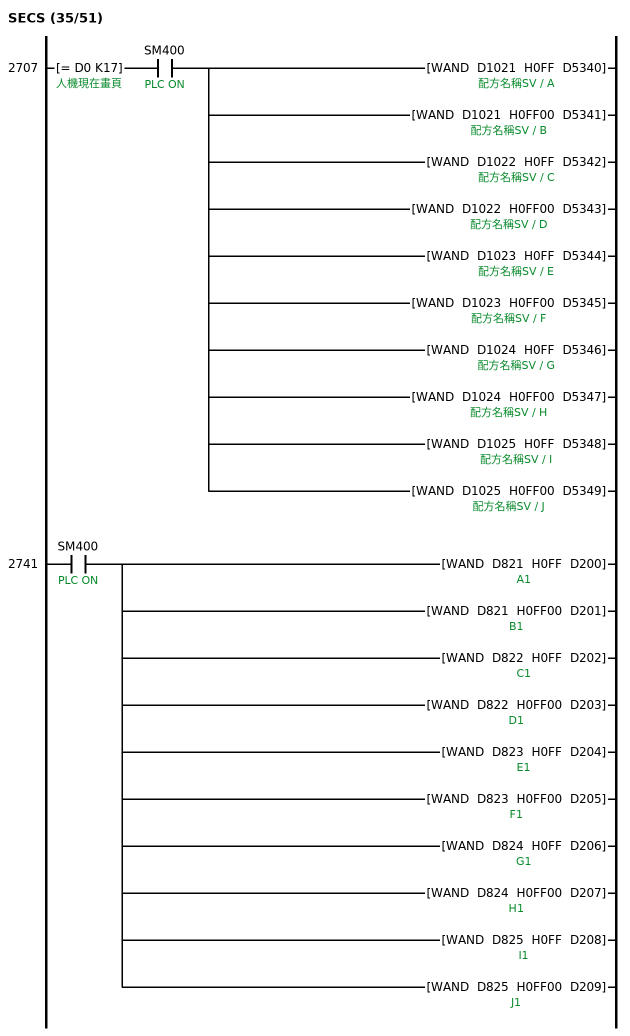
2707  LD=     D0 K17  ; 人機現在畫頁
      AND     SM400  ; PLC ON
      WAND    D1021 H0FF D5340  ; A
      WAND    D1021 H0FF00 D5341  ; B
      WAND    D1022 H0FF D5342  ; 配方名稱SV / C
      WAND    D1022 H0FF00 D5343  ; D
      WAND    D1023 H0FF D5344  ; 配方名稱SV / E
      WAND    D1023 H0FF00 D5345  ; F
      WAND    D1024 H0FF D5346  ; 配方名稱SV / G
      WAND    D1024 H0FF00 D5347  ; H
      WAND    D1025 H0FF D5348  ; 配方名稱SV / I
      WAND    D1025 H0FF00 D5349  ; J
2741  LD      SM400  ; PLC ON
      WAND    D821 H0FF D200  ; A1
      WAND    D821 H0FF00 D201  ; B1
      WAND    D822 H0FF D202  ; C1
      WAND    D822 H0FF00 D203  ; D1
      WAND    D823 H0FF D204  ; E1
      WAND    D823 H0FF00 D205  ; F1
      WAND    D824 H0FF D206  ; G1
      WAND    D824 H0FF00 D207  ; H1
      WAND    D825 H0FF D208  ; I1
      WAND    D825 H0FF00 D209  ; J1
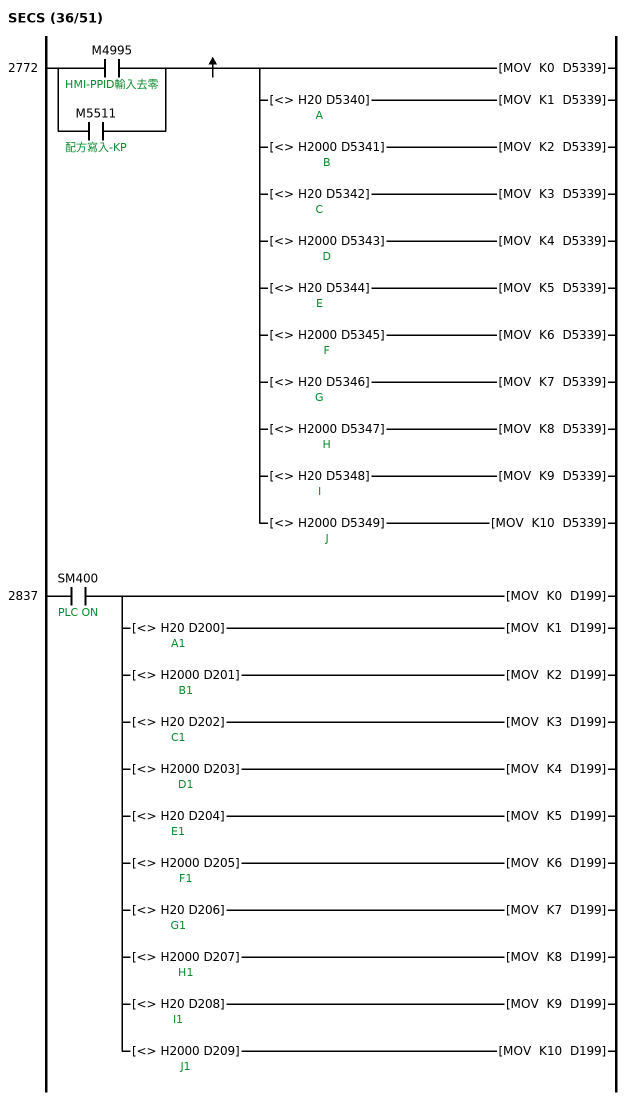
2772  LD      M4995  ; HMI-PPID輸入去零
      OR      M5511  ; 配方寫入-KP
      MEP
      MOV     K0 D5339
      MPS
      AND<>   H20 D5340  ; A
      MOV     K1 D5339
      MRD
      AND<>   H2000 D5341  ; B
      MOV     K2 D5339
      MRD
      AND<>   H20 D5342  ; C
      MOV     K3 D5339
      MRD
      AND<>   H2000 D5343  ; D
      MOV     K4 D5339
      MRD
      AND<>   H20 D5344  ; E
      MOV     K5 D5339
      MRD
      AND<>   H2000 D5345  ; F
      MOV     K6 D5339
      MRD
      AND<>   H20 D5346  ; G
      MOV     K7 D5339
      MRD
      AND<>   H2000 D5347  ; H
      MOV     K8 D5339
      MRD
      AND<>   H20 D5348  ; I
      MOV     K9 D5339
      MPP
      AND<>   H2000 D5349  ; J
      MOV     K10 D5339
2837  LD      SM400  ; PLC ON
      MOV     K0 D199
      MPS
      AND<>   H20 D200  ; A1
      MOV     K1 D199
      MRD
      AND<>   H2000 D201  ; B1
      MOV     K2 D199
      MRD
      AND<>   H20 D202  ; C1
      MOV     K3 D199
      MRD
      AND<>   H2000 D203  ; D1
      MOV     K4 D199
      MRD
      AND<>   H20 D204  ; E1
      MOV     K5 D199
      MRD
      AND<>   H2000 D205  ; F1
      MOV     K6 D199
      MRD
      AND<>   H20 D206  ; G1
      MOV     K7 D199
      MRD
      AND<>   H2000 D207  ; H1
      MOV     K8 D199
      MRD
      AND<>   H20 D208  ; I1
      MOV     K9 D199
      MPP
      AND<>   H2000 D209  ; J1
      MOV     K10 D199
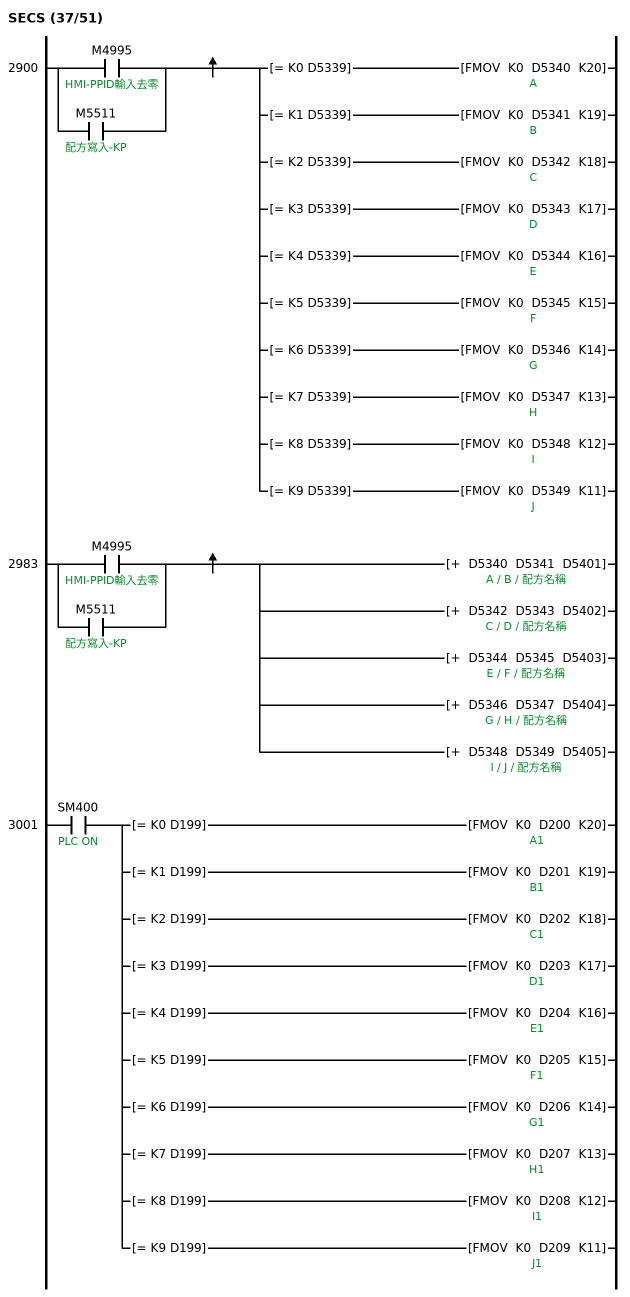
2900  LD      M4995  ; HMI-PPID輸入去零
      OR      M5511  ; 配方寫入-KP
      MEP
      MPS
      AND=    K0 D5339
      FMOV    K0 D5340 K20
      MRD
      AND=    K1 D5339
      FMOV    K0 D5341 K19
      MRD
      AND=    K2 D5339
      FMOV    K0 D5342 K18
      MRD
      AND=    K3 D5339
      FMOV    K0 D5343 K17
      MRD
      AND=    K4 D5339
      FMOV    K0 D5344 K16
      MRD
      AND=    K5 D5339
      FMOV    K0 D5345 K15
      MRD
      AND=    K6 D5339
      FMOV    K0 D5346 K14
      MRD
      AND=    K7 D5339
      FMOV    K0 D5347 K13
      MRD
      AND=    K8 D5339
      FMOV    K0 D5348 K12
      MPP
      AND=    K9 D5339
      FMOV    K0 D5349 K11
2983  LD      M4995  ; HMI-PPID輸入去零
      OR      M5511  ; 配方寫入-KP
      MEP
      +       D5340 D5341 D5401
      +       D5342 D5343 D5402  ; 配方名稱
      +       D5344 D5345 D5403  ; 配方名稱
      +       D5346 D5347 D5404  ; 配方名稱
      +       D5348 D5349 D5405  ; 配方名稱
3001  LD      SM400  ; PLC ON
      MPS
      AND=    K0 D199
      FMOV    K0 D200 K20
      MRD
      AND=    K1 D199
      FMOV    K0 D201 K19
      MRD
      AND=    K2 D199
      FMOV    K0 D202 K18
      MRD
      AND=    K3 D199
      FMOV    K0 D203 K17
      MRD
      AND=    K4 D199
      FMOV    K0 D204 K16
      MRD
      AND=    K5 D199
      FMOV    K0 D205 K15
      MRD
      AND=    K6 D199
      FMOV    K0 D206 K14
      MRD
      AND=    K7 D199
      FMOV    K0 D207 K13
      MRD
      AND=    K8 D199
      FMOV    K0 D208 K12
      MPP
      AND=    K9 D199
      FMOV    K0 D209 K11
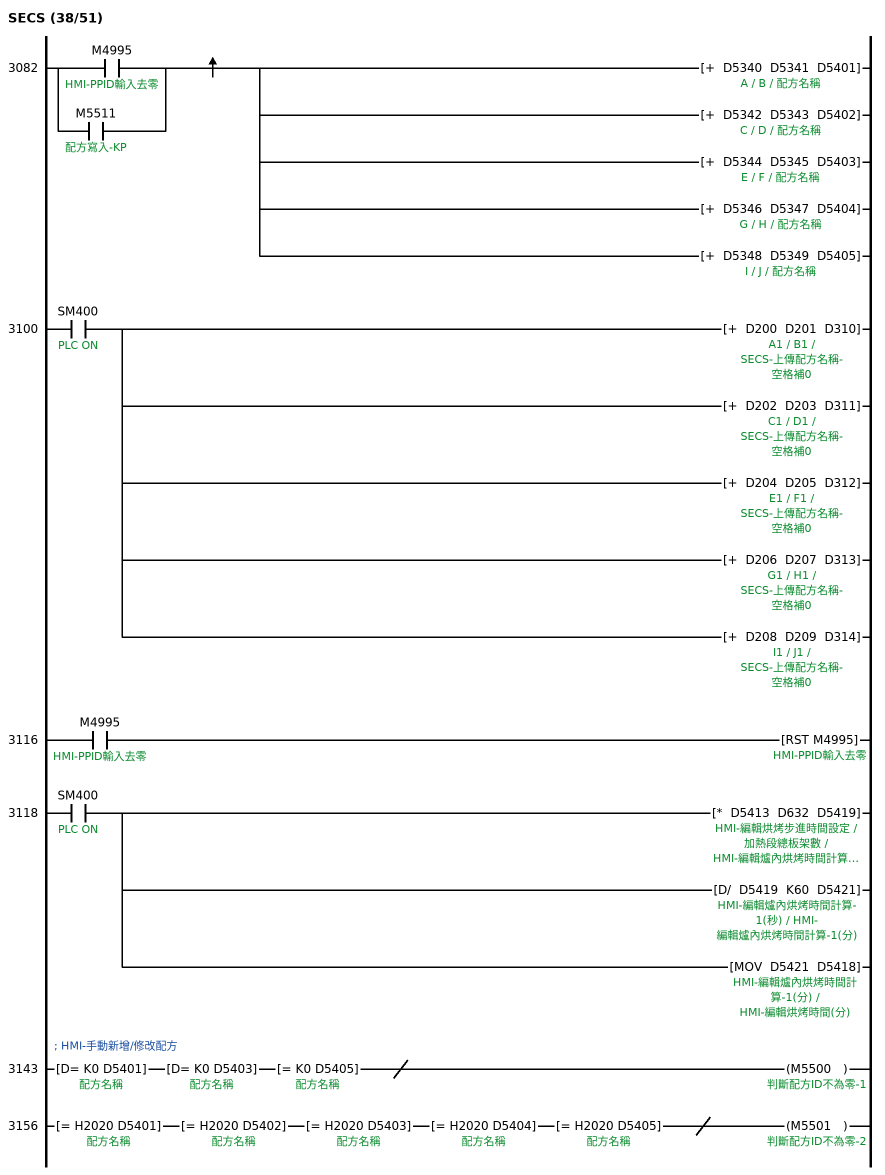
3082  LD      M4995  ; HMI-PPID輸入去零
      OR      M5511  ; 配方寫入-KP
      MEP
      +       D5340 D5341 D5401
      +       D5342 D5343 D5402
      +       D5344 D5345 D5403
      +       D5346 D5347 D5404
      +       D5348 D5349 D5405
3100  LD      SM400  ; PLC ON
      +       D200 D201 D310  ; SECS-上傳配方名稱-空格補0
      +       D202 D203 D311  ; SECS-上傳配方名稱-空格補0
      +       D204 D205 D312  ; SECS-上傳配方名稱-空格補0
      +       D206 D207 D313  ; SECS-上傳配方名稱-空格補0
      +       D208 D209 D314  ; SECS-上傳配方名稱-空格補0
3116  LD      M4995  ; HMI-PPID輸入去零
      RST     M4995  ; HMI-PPID輸入去零
3118  LD      SM400  ; PLC ON
      *       D5413 D632 D5419  ; HMI-編輯烘烤步進時間設定 / 加熱段總板架數 / HMI-編輯爐內烘烤時間計算-1(秒)
      D/      D5419 K60 D5421  ; HMI-編輯爐內烘烤時間計算-1(分)
      MOV     D5421 D5418  ; HMI-編輯烘烤時間(分)
; HMI-手動新增/修改配方
3143  LDD=    K0 D5401  ; 配方名稱
      ANDD=   K0 D5403  ; 配方名稱
      AND=    K0 D5405  ; 配方名稱
      INV
      OUT     M5500  ; 判斷配方ID不為零-1
3156  LD=     H2020 D5401  ; 配方名稱
      AND=    H2020 D5402  ; 配方名稱
      AND=    H2020 D5403  ; 配方名稱
      AND=    H2020 D5404  ; 配方名稱
      AND=    H2020 D5405  ; 配方名稱
      INV
      OUT     M5501  ; 判斷配方ID不為零-2
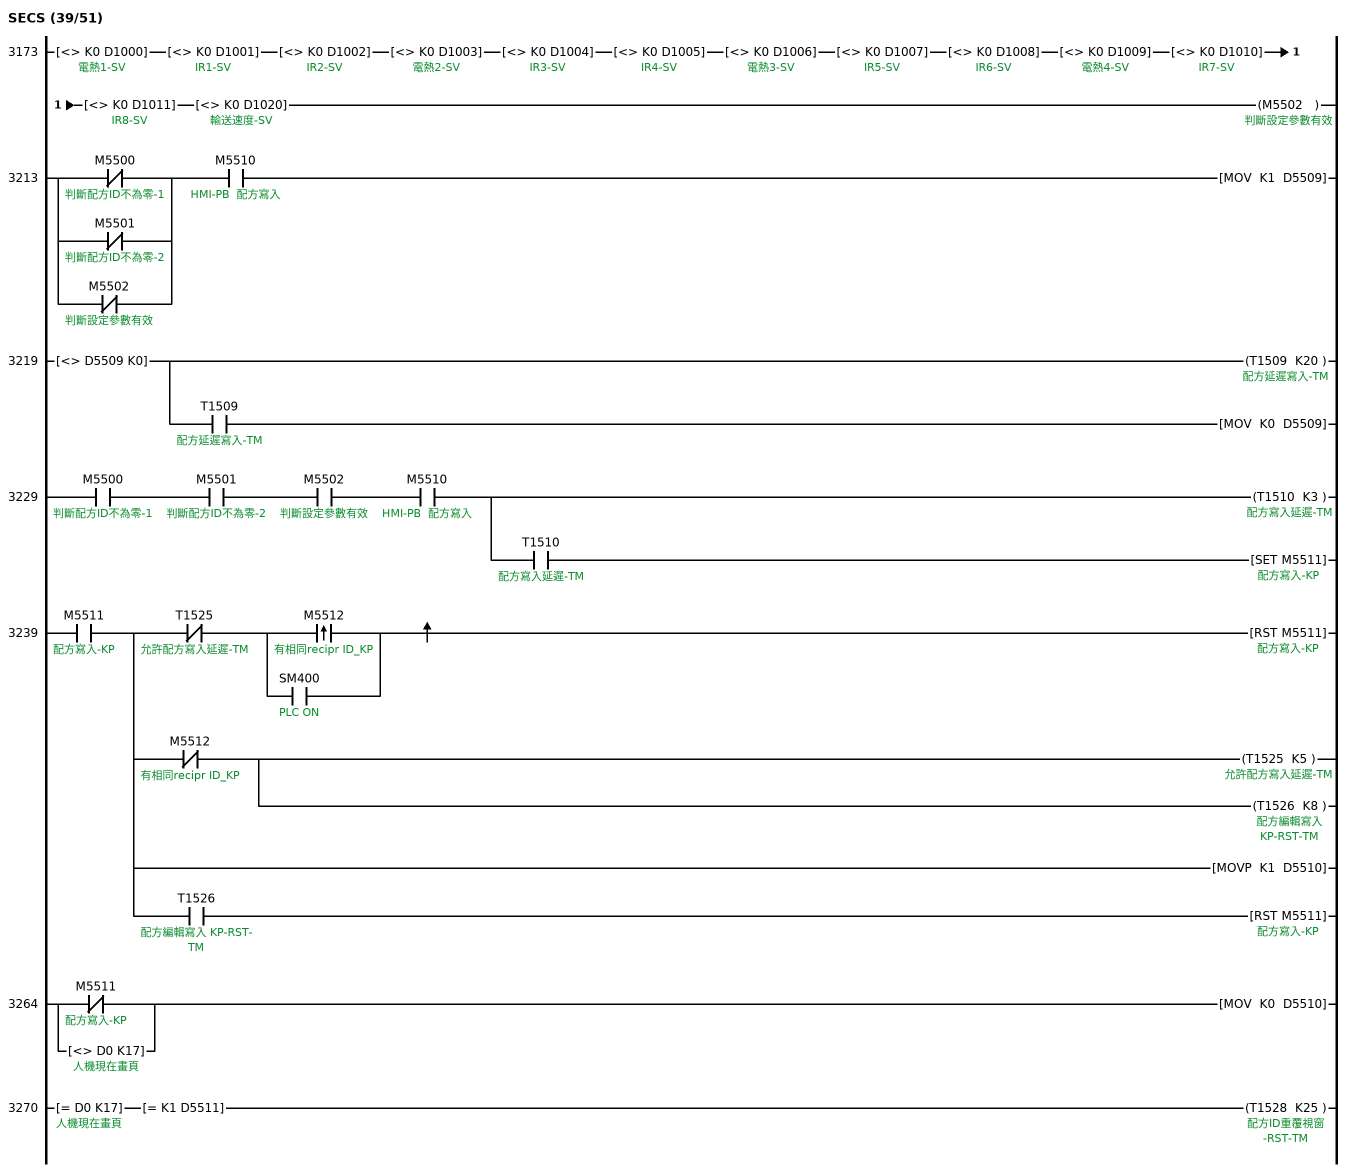
3173  LD<>    K0 D1000  ; 電熱1-SV
      AND<>   K0 D1001  ; IR1-SV
      AND<>   K0 D1002  ; IR2-SV
      AND<>   K0 D1003  ; 電熱2-SV
      AND<>   K0 D1004  ; IR3-SV
      AND<>   K0 D1005  ; IR4-SV
      AND<>   K0 D1006  ; 電熱3-SV
      AND<>   K0 D1007  ; IR5-SV
      AND<>   K0 D1008  ; IR6-SV
      AND<>   K0 D1009  ; 電熱4-SV
      AND<>   K0 D1010  ; IR7-SV
      AND<>   K0 D1011  ; IR8-SV
      AND<>   K0 D1020  ; 輸送速度-SV
      OUT     M5502  ; 判斷設定參數有效
3213  LDI     M5500  ; 判斷配方ID不為零-1
      ORI     M5501  ; 判斷配方ID不為零-2
      ORI     M5502  ; 判斷設定參數有效
      AND     M5510  ; HMI-PB  配方寫入
      MOV     K1 D5509
3219  LD<>    D5509 K0
      OUT     T1509 K20  ; 配方延遲寫入-TM
      AND     T1509  ; 配方延遲寫入-TM
      MOV     K0 D5509
3229  LD      M5500  ; 判斷配方ID不為零-1
      AND     M5501  ; 判斷配方ID不為零-2
      AND     M5502  ; 判斷設定參數有效
      AND     M5510  ; HMI-PB  配方寫入
      OUT     T1510 K3  ; 配方寫入延遲-TM
      AND     T1510  ; 配方寫入延遲-TM
      SET     M5511  ; 配方寫入-KP
3239  LD      M5511  ; 配方寫入-KP
      MPS
      ANI     T1525  ; 允許配方寫入延遲-TM
      LDP     M5512  ; 有相同recipr ID_KP
      OR      SM400  ; PLC ON
      ANB
      MEP
      RST     M5511  ; 配方寫入-KP
      MRD
      ANI     M5512  ; 有相同recipr ID_KP
      OUT     T1525 K5  ; 允許配方寫入延遲-TM
      OUT     T1526 K8  ; 配方編輯寫入 KP-RST-TM
      MPP
      MOVP    K1 D5510
      AND     T1526  ; 配方編輯寫入 KP-RST-TM
      RST     M5511  ; 配方寫入-KP
3264  LDI     M5511  ; 配方寫入-KP
      OR<>    D0 K17  ; 人機現在畫頁
      MOV     K0 D5510
3270  LD=     D0 K17  ; 人機現在畫頁
      AND=    K1 D5511
      OUT     T1528 K25  ; 配方ID重覆視窗  -RST-TM
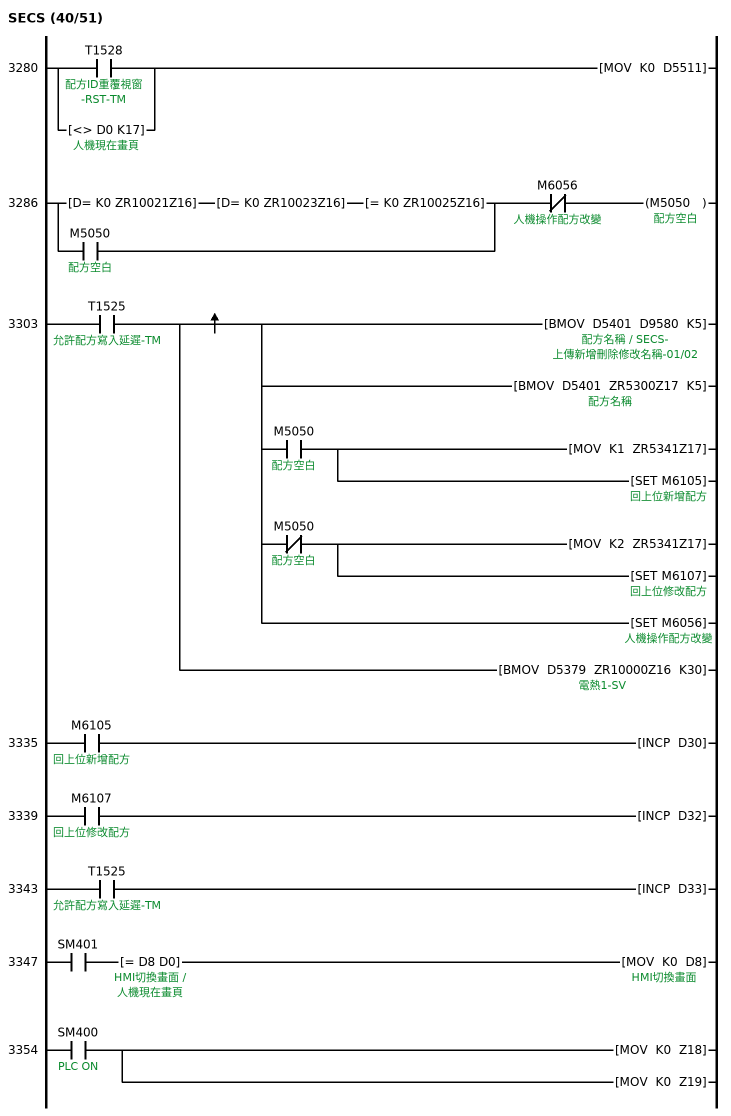
3280  LD      T1528  ; 配方ID重覆視窗  -RST-TM
      OR<>    D0 K17  ; 人機現在畫頁
      MOV     K0 D5511
3286  LDD=    K0 ZR10021Z16
      ANDD=   K0 ZR10023Z16
      AND=    K0 ZR10025Z16
      OR      M5050  ; 配方空白
      ANI     M6056  ; 人機操作配方改變
      OUT     M5050  ; 配方空白
3303  LD      T1525  ; 允許配方寫入延遲-TM
      MPS
      MEP
      BMOV    D5401 D9580 K5  ; SECS-上傳新增刪除修改名稱-01/02
      BMOV    D5401 ZR5300Z17 K5
      MPS
      AND     M5050  ; 配方空白
      MOV     K1 ZR5341Z17
      SET     M6105  ; 回上位新增配方
      MRD
      ANI     M5050  ; 配方空白
      MOV     K2 ZR5341Z17
      SET     M6107  ; 回上位修改配方
      MPP
      SET     M6056  ; 人機操作配方改變
      MPP
      BMOV    D5379 ZR10000Z16 K30
3335  LD      M6105  ; 回上位新增配方
      INCP    D30
3339  LD      M6107  ; 回上位修改配方
      INCP    D32
3343  LD      T1525  ; 允許配方寫入延遲-TM
      INCP    D33
3347  LD      SM401
      AND=    D8 D0  ; HMI切換畫面 / 人機現在畫頁
      MOV     K0 D8
3354  LD      SM400  ; PLC ON
      MOV     K0 Z18
      MOV     K0 Z19
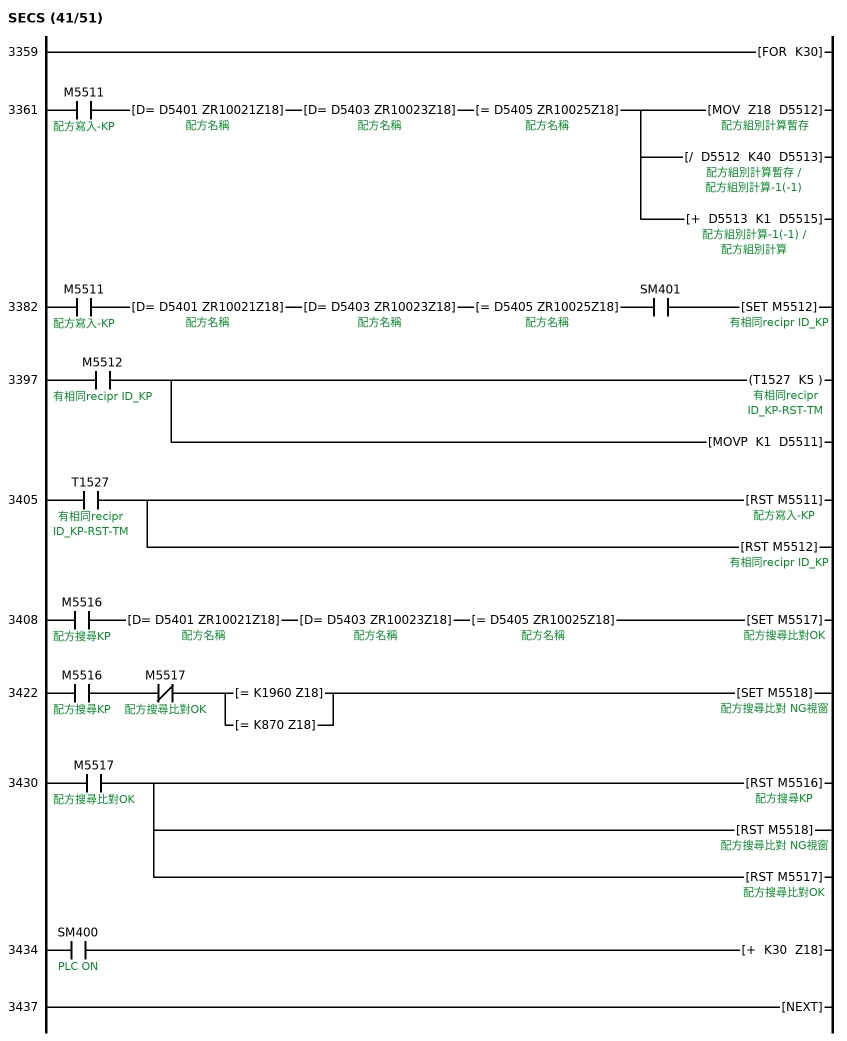
3359  FOR     K30
3361  LD      M5511  ; 配方寫入-KP
      ANDD=   D5401 ZR10021Z18  ; 配方名稱
      ANDD=   D5403 ZR10023Z18  ; 配方名稱
      AND=    D5405 ZR10025Z18  ; 配方名稱
      MOV     Z18 D5512  ; 配方組別計算暫存
      /       D5512 K40 D5513  ; 配方組別計算-1(-1)
      +       D5513 K1 D5515  ; 配方組別計算
3382  LD      M5511  ; 配方寫入-KP
      ANDD=   D5401 ZR10021Z18  ; 配方名稱
      ANDD=   D5403 ZR10023Z18  ; 配方名稱
      AND=    D5405 ZR10025Z18  ; 配方名稱
      AND     SM401
      SET     M5512  ; 有相同recipr ID_KP
3397  LD      M5512  ; 有相同recipr ID_KP
      OUT     T1527 K5  ; 有相同recipr ID_KP-RST-TM
      MOVP    K1 D5511
3405  LD      T1527  ; 有相同recipr ID_KP-RST-TM
      RST     M5511  ; 配方寫入-KP
      RST     M5512  ; 有相同recipr ID_KP
3408  LD      M5516  ; 配方搜尋KP
      ANDD=   D5401 ZR10021Z18  ; 配方名稱
      ANDD=   D5403 ZR10023Z18  ; 配方名稱
      AND=    D5405 ZR10025Z18  ; 配方名稱
      SET     M5517  ; 配方搜尋比對OK
3422  LD      M5516  ; 配方搜尋KP
      ANI     M5517  ; 配方搜尋比對OK
      LD=     K1960 Z18
      OR=     K870 Z18
      ANB
      SET     M5518  ; 配方搜尋比對 NG視窗
3430  LD      M5517  ; 配方搜尋比對OK
      RST     M5516  ; 配方搜尋KP
      RST     M5518  ; 配方搜尋比對 NG視窗
      RST     M5517  ; 配方搜尋比對OK
3434  LD      SM400  ; PLC ON
      +       K30 Z18
3437  NEXT
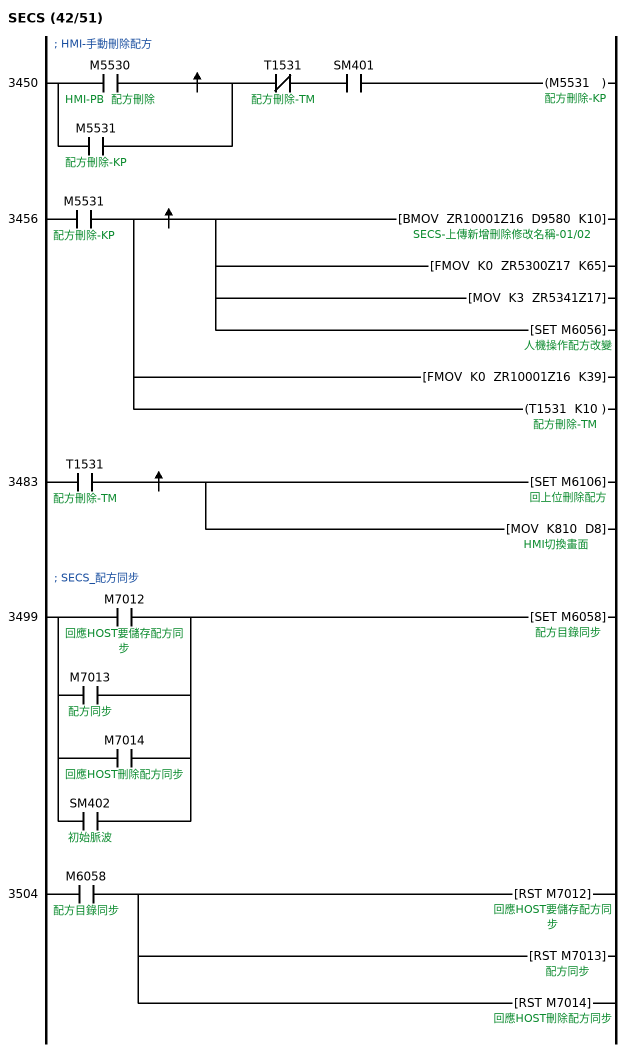
; HMI-手動刪除配方
3450  LD      M5530  ; HMI-PB  配方刪除
      MEP
      OR      M5531  ; 配方刪除-KP
      ANI     T1531  ; 配方刪除-TM
      AND     SM401
      OUT     M5531  ; 配方刪除-KP
3456  LD      M5531  ; 配方刪除-KP
      MPS
      MEP
      BMOV    ZR10001Z16 D9580 K10
      FMOV    K0 ZR5300Z17 K65
      MOV     K3 ZR5341Z17
      SET     M6056  ; 人機操作配方改變
      MPP
      FMOV    K0 ZR10001Z16 K39
      OUT     T1531 K10  ; 配方刪除-TM
3483  LD      T1531  ; 配方刪除-TM
      MEP
      SET     M6106  ; 回上位刪除配方
      MOV     K810 D8
; SECS_配方同步
3499  LD      M7012  ; 回應HOST要儲存配方同步
      OR      M7013  ; 配方同步
      OR      M7014  ; 回應HOST刪除配方同步
      OR      SM402  ; 初始脈波
      SET     M6058  ; 配方目錄同步
3504  LD      M6058  ; 配方目錄同步
      RST     M7012  ; 回應HOST要儲存配方同步
      RST     M7013  ; 配方同步
      RST     M7014  ; 回應HOST刪除配方同步
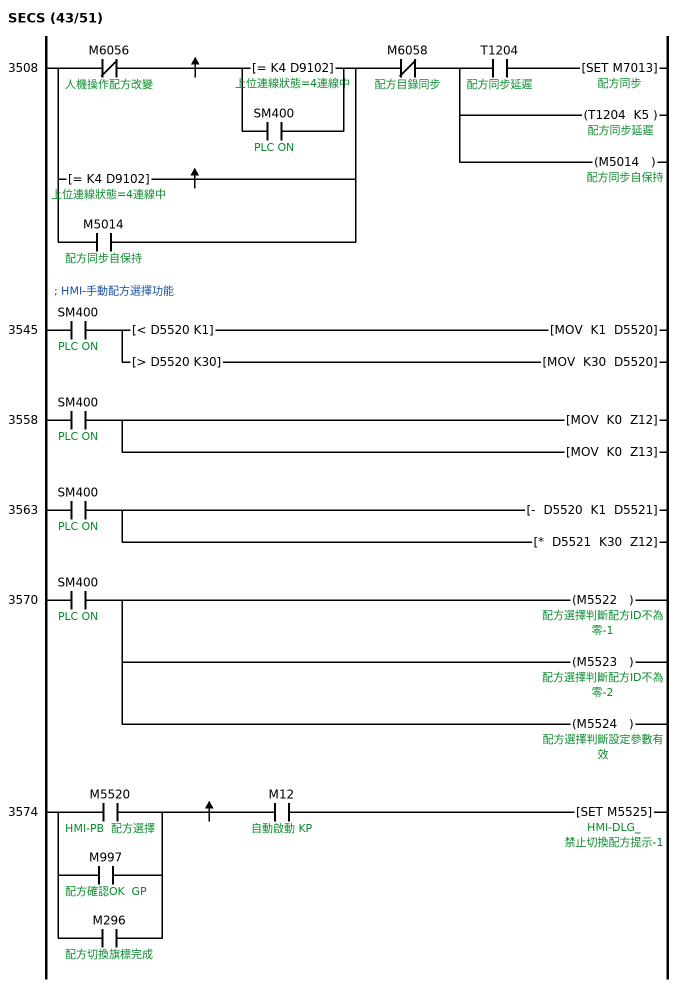
3508  LDI     M6056  ; 人機操作配方改變
      MEP
      LD=     K4 D9102  ; 上位連線狀態=4連線中
      OR      SM400  ; PLC ON
      ANB
      LD=     K4 D9102  ; 上位連線狀態=4連線中
      MEP
      ORB
      OR      M5014  ; 配方同步自保持
      ANI     M6058  ; 配方目錄同步
      MPS
      AND     T1204  ; 配方同步延遲
      SET     M7013  ; 配方同步
      MPP
      OUT     T1204 K5  ; 配方同步延遲
      OUT     M5014  ; 配方同步自保持
; HMI-手動配方選擇功能
3545  LD      SM400  ; PLC ON
      MPS
      AND<    D5520 K1
      MOV     K1 D5520
      MPP
      AND>    D5520 K30
      MOV     K30 D5520
3558  LD      SM400  ; PLC ON
      MOV     K0 Z12
      MOV     K0 Z13
3563  LD      SM400  ; PLC ON
      -       D5520 K1 D5521
      *       D5521 K30 Z12
3570  LD      SM400  ; PLC ON
      OUT     M5522  ; 配方選擇判斷配方ID不為零-1
      OUT     M5523  ; 配方選擇判斷配方ID不為零-2
      OUT     M5524  ; 配方選擇判斷設定參數有效
3574  LD      M5520  ; HMI-PB  配方選擇
      OR      M997  ; 配方確認OK  GP
      OR      M296  ; 配方切換旗標完成
      MEP
      AND     M12  ; 自動啟動 KP
      SET     M5525  ; HMI-DLG_禁止切換配方提示-1
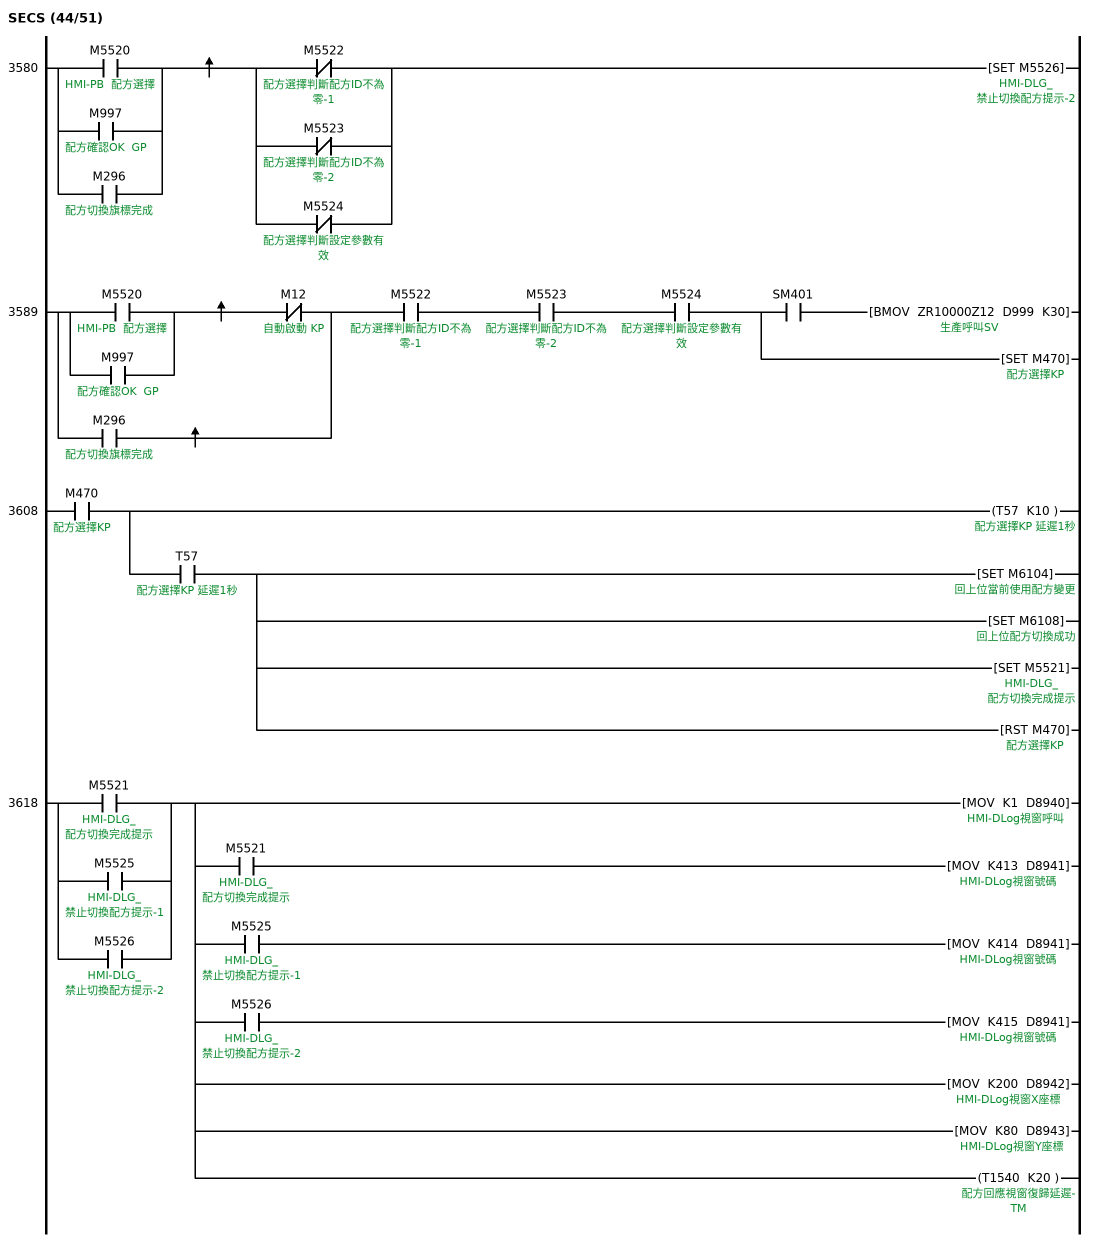
3580  LD      M5520  ; HMI-PB  配方選擇
      OR      M997  ; 配方確認OK  GP
      OR      M296  ; 配方切換旗標完成
      MEP
      LDI     M5522  ; 配方選擇判斷配方ID不為零-1
      ORI     M5523  ; 配方選擇判斷配方ID不為零-2
      ORI     M5524  ; 配方選擇判斷設定參數有效
      ANB
      SET     M5526  ; HMI-DLG_禁止切換配方提示-2
3589  LD      M5520  ; HMI-PB  配方選擇
      OR      M997  ; 配方確認OK  GP
      MEP
      ANI     M12  ; 自動啟動 KP
      LD      M296  ; 配方切換旗標完成
      MEP
      ORB
      AND     M5522  ; 配方選擇判斷配方ID不為零-1
      AND     M5523  ; 配方選擇判斷配方ID不為零-2
      AND     M5524  ; 配方選擇判斷設定參數有效
      MPS
      AND     SM401
      BMOV    ZR10000Z12 D999 K30
      MPP
      SET     M470  ; 配方選擇KP
3608  LD      M470  ; 配方選擇KP
      OUT     T57 K10  ; 配方選擇KP 延遲1秒
      AND     T57  ; 配方選擇KP 延遲1秒
      SET     M6104  ; 回上位當前使用配方變更
      SET     M6108  ; 回上位配方切換成功
      SET     M5521  ; HMI-DLG_配方切換完成提示
      RST     M470  ; 配方選擇KP
3618  LD      M5521  ; HMI-DLG_配方切換完成提示
      OR      M5525  ; HMI-DLG_禁止切換配方提示-1
      OR      M5526  ; HMI-DLG_禁止切換配方提示-2
      MOV     K1 D8940  ; HMI-DLog視窗呼叫
      MPS
      AND     M5521  ; HMI-DLG_配方切換完成提示
      MOV     K413 D8941  ; HMI-DLog視窗號碼
      MRD
      AND     M5525  ; HMI-DLG_禁止切換配方提示-1
      MOV     K414 D8941
      MRD
      AND     M5526  ; HMI-DLG_禁止切換配方提示-2
      MOV     K415 D8941
      MPP
      MOV     K200 D8942  ; HMI-DLog視窗X座標
      MOV     K80 D8943  ; HMI-DLog視窗Y座標
      OUT     T1540 K20  ; 配方回應視窗復歸延遲-TM
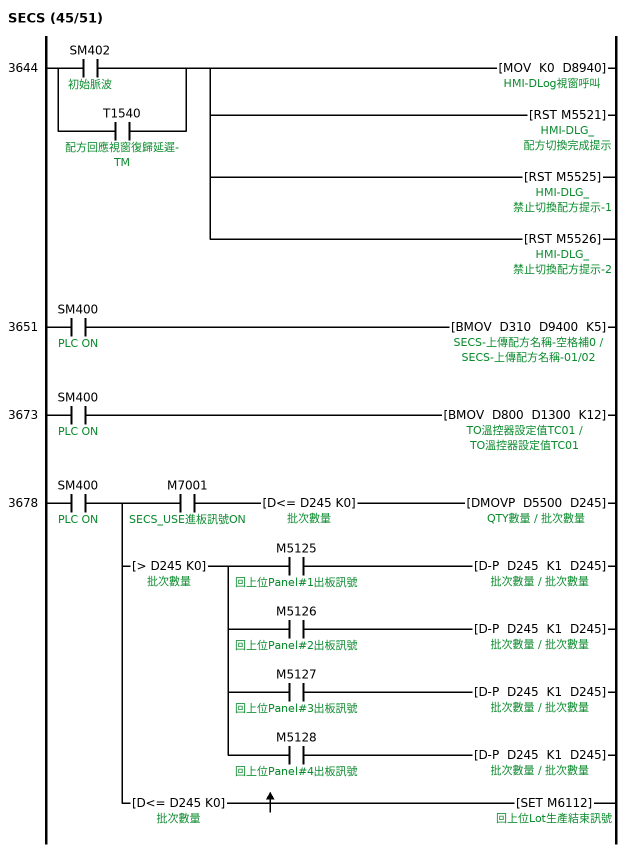
3644  LD      SM402  ; 初始脈波
      OR      T1540  ; 配方回應視窗復歸延遲-TM
      MOV     K0 D8940
      RST     M5521  ; HMI-DLG_配方切換完成提示
      RST     M5525  ; HMI-DLG_禁止切換配方提示-1
      RST     M5526  ; HMI-DLG_禁止切換配方提示-2
3651  LD      SM400  ; PLC ON
      BMOV    D310 D9400 K5  ; SECS-上傳配方名稱-01/02
        [note] D9400_上報SECS目前使用PPID名稱
3673  LD      SM400  ; PLC ON
      BMOV    D800 D1300 K12  ; TO溫控器設定值TC01
3678  LD      SM400  ; PLC ON
      MPS
      AND     M7001  ; SECS_USE進板訊號ON
      ANDD<=  D245 K0  ; 批次數量
      DMOVP   D5500 D245
      MRD
      AND>    D245 K0  ; 批次數量
      MPS
      AND     M5125  ; 回上位Panel#1出板訊號
      D-P     D245 K1 D245
      MRD
      AND     M5126  ; 回上位Panel#2出板訊號
      D-P     D245 K1 D245
      MRD
      AND     M5127  ; 回上位Panel#3出板訊號
      D-P     D245 K1 D245
      MPP
      AND     M5128  ; 回上位Panel#4出板訊號
      D-P     D245 K1 D245
      MPP
      ANDD<=  D245 K0  ; 批次數量
      MEP
      SET     M6112  ; 回上位Lot生產結束訊號
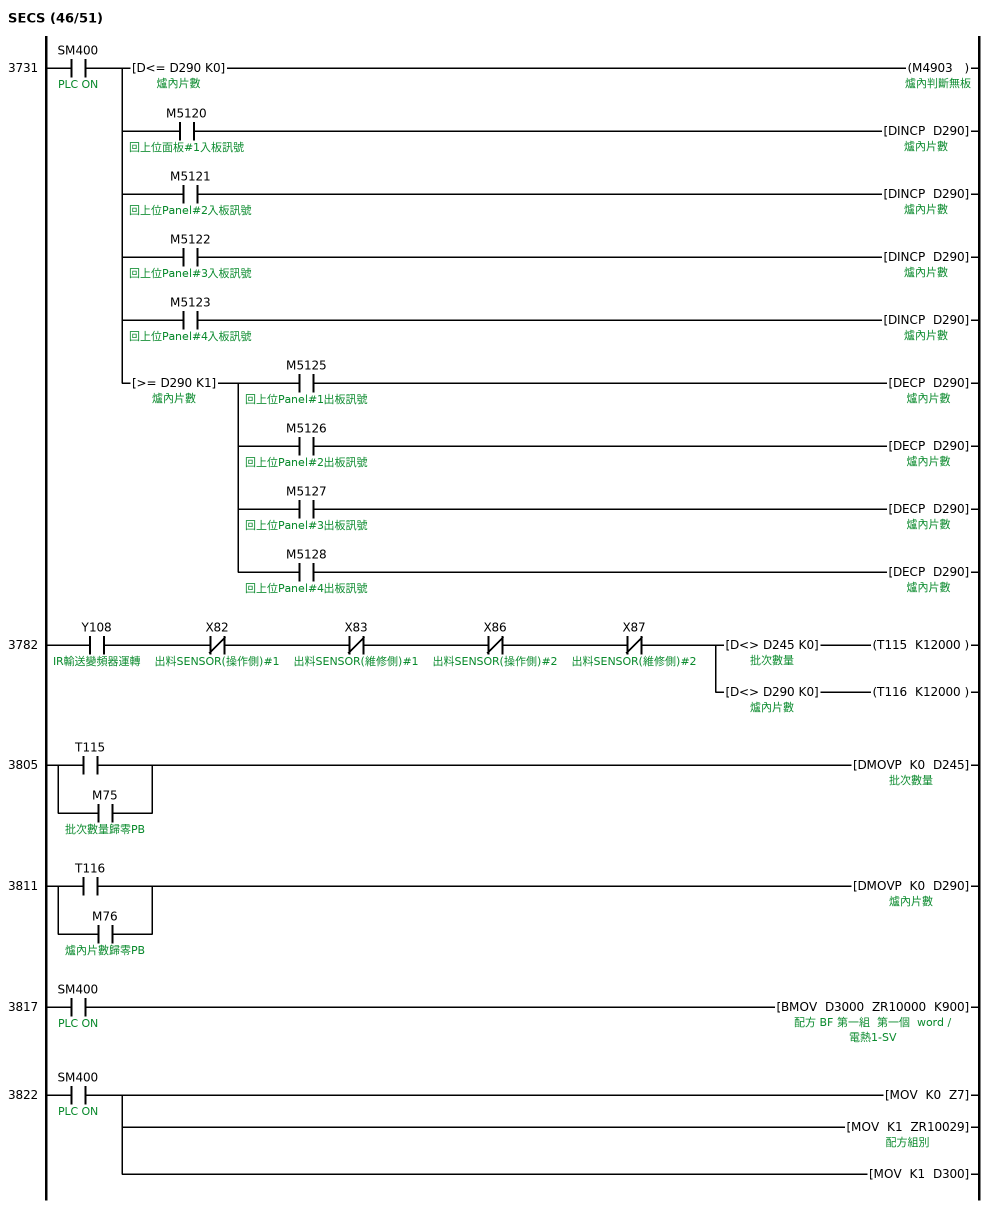
3731  LD      SM400  ; PLC ON
      MPS
      ANDD<=  D290 K0  ; 爐內片數
      OUT     M4903  ; 爐內判斷無板
      MRD
      AND     M5120  ; 回上位面板#1入板訊號
      DINCP   D290
      MRD
      AND     M5121  ; 回上位Panel#2入板訊號
      DINCP   D290
      MRD
      AND     M5122  ; 回上位Panel#3入板訊號
      DINCP   D290
      MRD
      AND     M5123  ; 回上位Panel#4入板訊號
      DINCP   D290
      MPP
      AND>=   D290 K1  ; 爐內片數
      MPS
      AND     M5125  ; 回上位Panel#1出板訊號
      DECP    D290
      MRD
      AND     M5126  ; 回上位Panel#2出板訊號
      DECP    D290
      MRD
      AND     M5127  ; 回上位Panel#3出板訊號
      DECP    D290
      MPP
      AND     M5128  ; 回上位Panel#4出板訊號
      DECP    D290
3782  LD      Y108  ; IR輸送變頻器運轉
      ANI     X82  ; 出料SENSOR(操作側)#1
      ANI     X83  ; 出料SENSOR(維修側)#1
      ANI     X86  ; 出料SENSOR(操作側)#2
      ANI     X87  ; 出料SENSOR(維修側)#2
      MPS
      ANDD<>  D245 K0  ; 批次數量
      OUT     T115 K12000
      MPP
      ANDD<>  D290 K0  ; 爐內片數
      OUT     T116 K12000
3805  LD      T115
      OR      M75  ; 批次數量歸零PB
      DMOVP   K0 D245
3811  LD      T116
      OR      M76  ; 爐內片數歸零PB
      DMOVP   K0 D290
3817  LD      SM400  ; PLC ON
      BMOV    D3000 ZR10000 K900  ; 配方 BF 第一組  第一個  word
3822  LD      SM400  ; PLC ON
      MOV     K0 Z7
      MOV     K1 ZR10029  ; 配方組別
      MOV     K1 D300
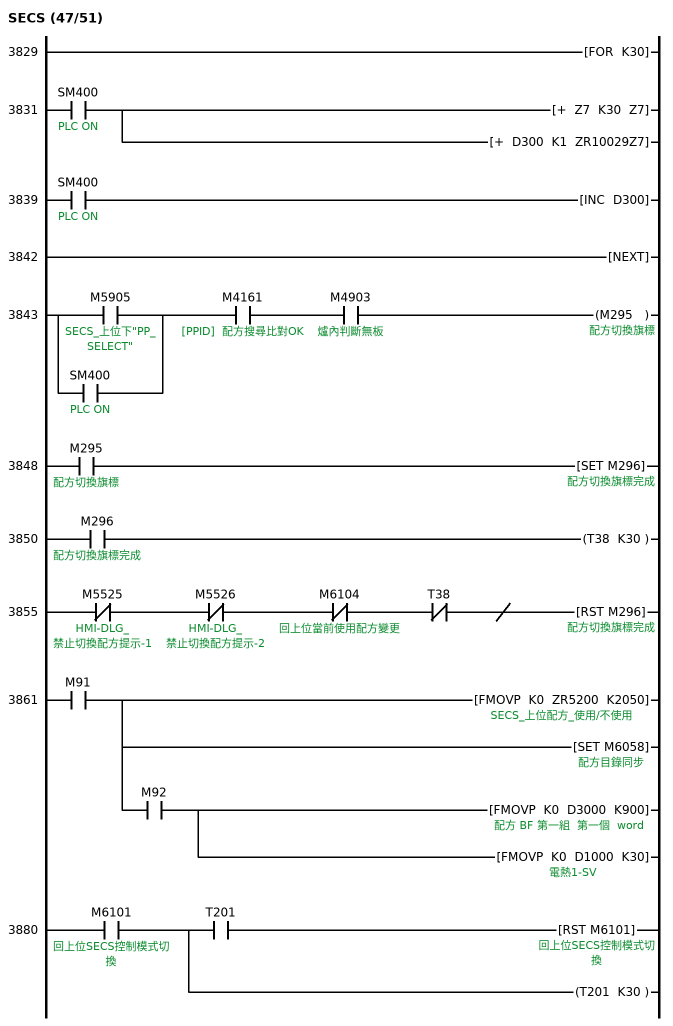
3829  FOR     K30
3831  LD      SM400  ; PLC ON
      +       Z7 K30 Z7
      +       D300 K1 ZR10029Z7
3839  LD      SM400  ; PLC ON
      INC     D300
3842  NEXT
3843  LD      M5905  ; SECS_上位下"PP_SELECT"
      OR      SM400  ; PLC ON
      AND     M4161  ; [PPID]  配方搜尋比對OK
      AND     M4903  ; 爐內判斷無板
      OUT     M295  ; 配方切換旗標
3848  LD      M295  ; 配方切換旗標
      SET     M296  ; 配方切換旗標完成
3850  LD      M296  ; 配方切換旗標完成
      OUT     T38 K30
3855  LDI     M5525  ; HMI-DLG_禁止切換配方提示-1
      ANI     M5526  ; HMI-DLG_禁止切換配方提示-2
      ANI     M6104  ; 回上位當前使用配方變更
      ANI     T38
      INV
      RST     M296  ; 配方切換旗標完成
3861  LD      M91
      FMOVP   K0 ZR5200 K2050  ; SECS_上位配方_使用/不使用
      SET     M6058  ; 配方目錄同步
      AND     M92
      FMOVP   K0 D3000 K900
      FMOVP   K0 D1000 K30
3880  LD      M6101  ; 回上位SECS控制模式切換
      MPS
      AND     T201
      RST     M6101  ; 回上位SECS控制模式切換
      MPP
      OUT     T201 K30
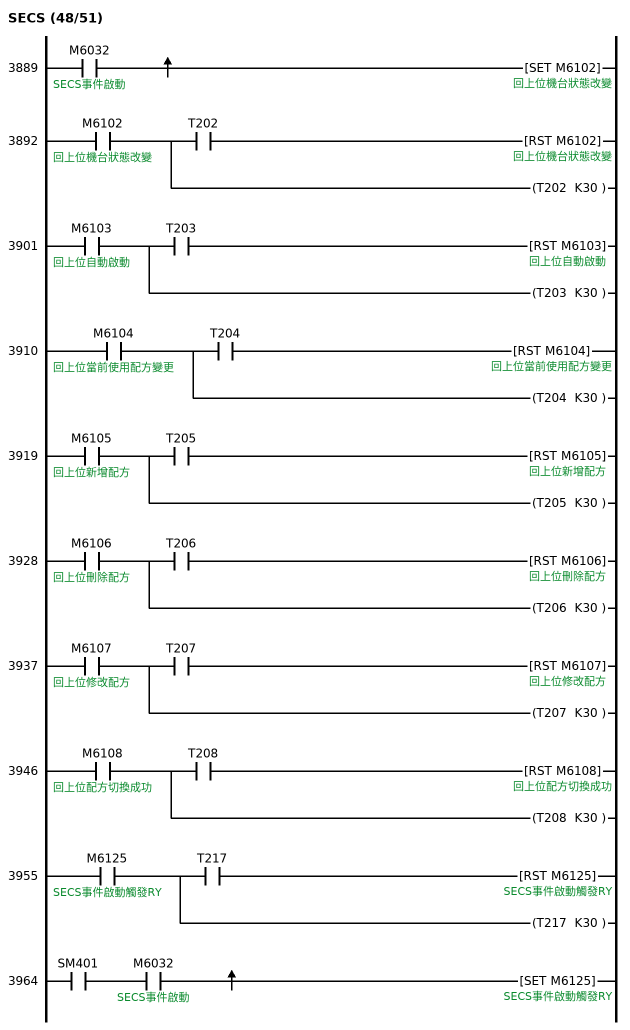
3889  LD      M6032  ; SECS事件啟動
      MEP
      SET     M6102  ; 回上位機台狀態改變
3892  LD      M6102  ; 回上位機台狀態改變
      MPS
      AND     T202
      RST     M6102  ; 回上位機台狀態改變
      MPP
      OUT     T202 K30
3901  LD      M6103  ; 回上位自動啟動
      MPS
      AND     T203
      RST     M6103  ; 回上位自動啟動
      MPP
      OUT     T203 K30
3910  LD      M6104  ; 回上位當前使用配方變更
      MPS
      AND     T204
      RST     M6104  ; 回上位當前使用配方變更
      MPP
      OUT     T204 K30
3919  LD      M6105  ; 回上位新增配方
      MPS
      AND     T205
      RST     M6105  ; 回上位新增配方
      MPP
      OUT     T205 K30
3928  LD      M6106  ; 回上位刪除配方
      MPS
      AND     T206
      RST     M6106  ; 回上位刪除配方
      MPP
      OUT     T206 K30
3937  LD      M6107  ; 回上位修改配方
      MPS
      AND     T207
      RST     M6107  ; 回上位修改配方
      MPP
      OUT     T207 K30
3946  LD      M6108  ; 回上位配方切換成功
      MPS
      AND     T208
      RST     M6108  ; 回上位配方切換成功
      MPP
      OUT     T208 K30
3955  LD      M6125  ; SECS事件啟動觸發RY
      MPS
      AND     T217
      RST     M6125  ; SECS事件啟動觸發RY
      MPP
      OUT     T217 K30
3964  LD      SM401
      AND     M6032  ; SECS事件啟動
      MEP
      SET     M6125  ; SECS事件啟動觸發RY
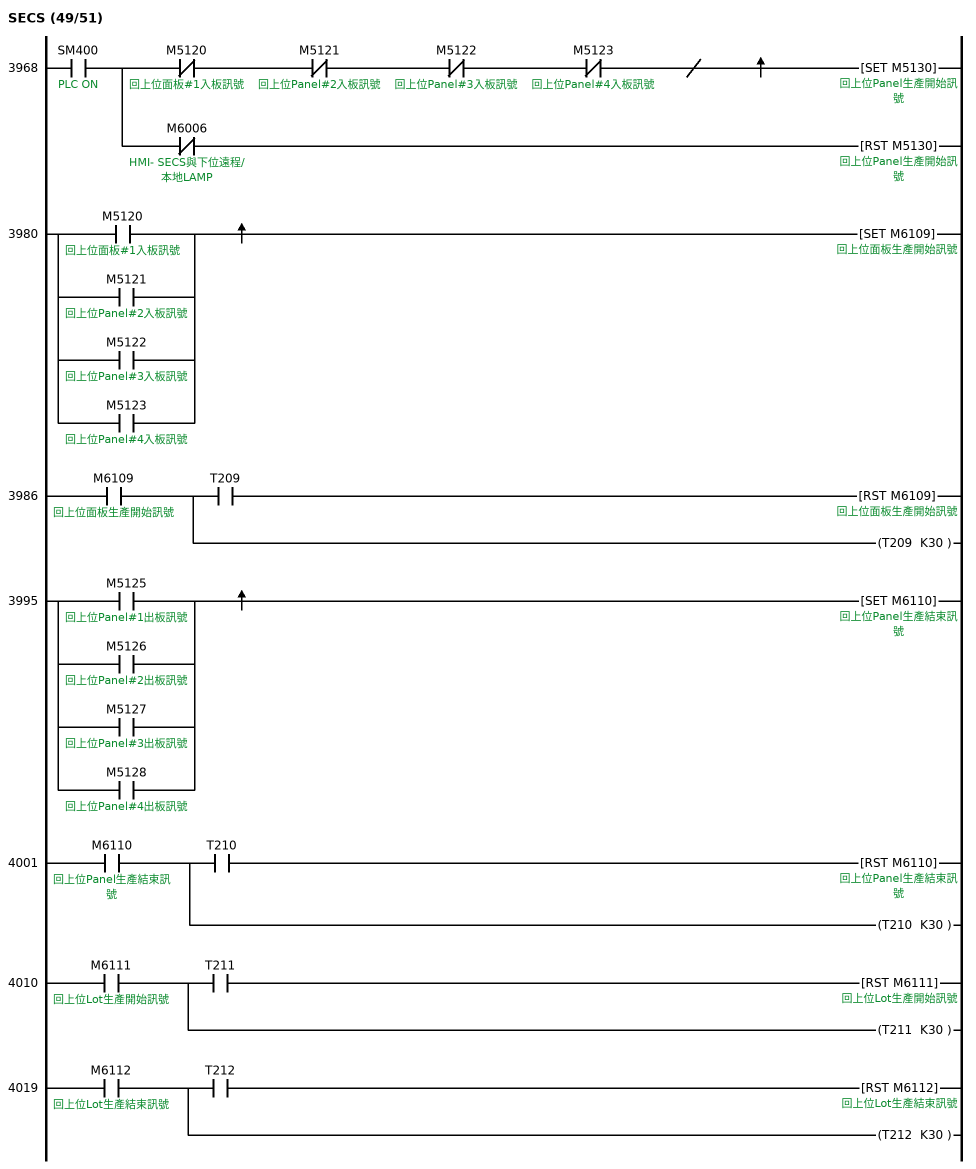
3968  LD      SM400  ; PLC ON
      MPS
      ANI     M5120  ; 回上位面板#1入板訊號
      ANI     M5121  ; 回上位Panel#2入板訊號
      ANI     M5122  ; 回上位Panel#3入板訊號
      ANI     M5123  ; 回上位Panel#4入板訊號
      INV
      MEP
      SET     M5130  ; 回上位Panel生產開始訊號
      MPP
      ANI     M6006  ; HMI- SECS與下位遠程/本地LAMP
      RST     M5130  ; 回上位Panel生產開始訊號
3980  LD      M5120  ; 回上位面板#1入板訊號
      OR      M5121  ; 回上位Panel#2入板訊號
      OR      M5122  ; 回上位Panel#3入板訊號
      OR      M5123  ; 回上位Panel#4入板訊號
      MEP
      SET     M6109  ; 回上位面板生產開始訊號
3986  LD      M6109  ; 回上位面板生產開始訊號
      MPS
      AND     T209
      RST     M6109  ; 回上位面板生產開始訊號
      MPP
      OUT     T209 K30
3995  LD      M5125  ; 回上位Panel#1出板訊號
      OR      M5126  ; 回上位Panel#2出板訊號
      OR      M5127  ; 回上位Panel#3出板訊號
      OR      M5128  ; 回上位Panel#4出板訊號
      MEP
      SET     M6110  ; 回上位Panel生產結束訊號
4001  LD      M6110  ; 回上位Panel生產結束訊號
      MPS
      AND     T210
      RST     M6110  ; 回上位Panel生產結束訊號
      MPP
      OUT     T210 K30
4010  LD      M6111  ; 回上位Lot生產開始訊號
      MPS
      AND     T211
      RST     M6111  ; 回上位Lot生產開始訊號
      MPP
      OUT     T211 K30
4019  LD      M6112  ; 回上位Lot生產結束訊號
      MPS
      AND     T212
      RST     M6112  ; 回上位Lot生產結束訊號
      MPP
      OUT     T212 K30
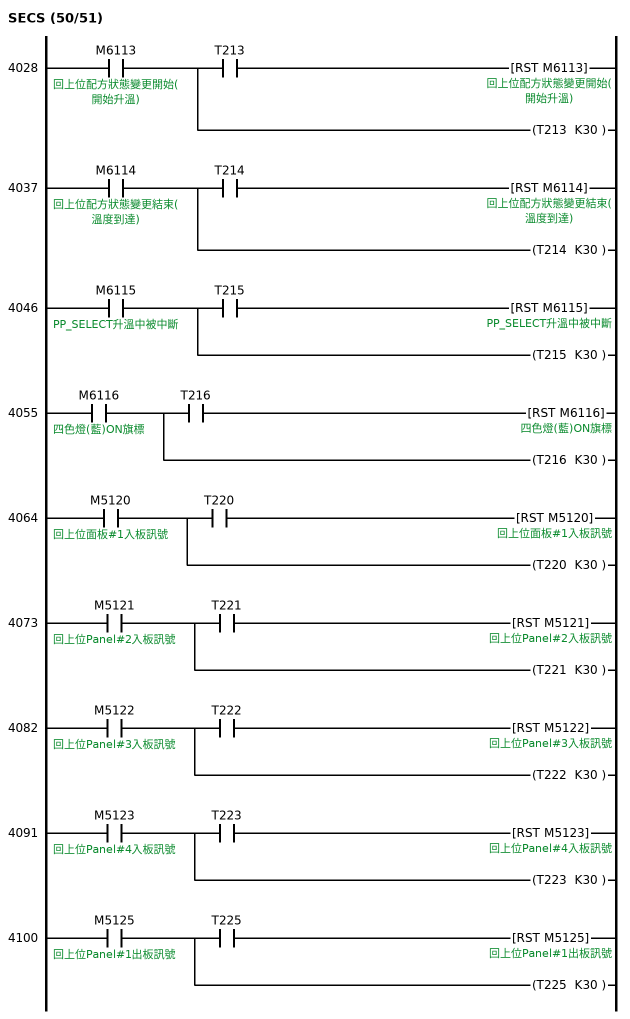
4028  LD      M6113  ; 回上位配方狀態變更開始(開始升溫)
      MPS
      AND     T213
      RST     M6113  ; 回上位配方狀態變更開始(開始升溫)
      MPP
      OUT     T213 K30
4037  LD      M6114  ; 回上位配方狀態變更結束(溫度到達)
      MPS
      AND     T214
      RST     M6114  ; 回上位配方狀態變更結束(溫度到達)
      MPP
      OUT     T214 K30
4046  LD      M6115  ; PP_SELECT升溫中被中斷
      MPS
      AND     T215
      RST     M6115  ; PP_SELECT升溫中被中斷
      MPP
      OUT     T215 K30
4055  LD      M6116  ; 四色燈(藍)ON旗標
      MPS
      AND     T216
      RST     M6116  ; 四色燈(藍)ON旗標
      MPP
      OUT     T216 K30
4064  LD      M5120  ; 回上位面板#1入板訊號
      MPS
      AND     T220
      RST     M5120  ; 回上位面板#1入板訊號
      MPP
      OUT     T220 K30
4073  LD      M5121  ; 回上位Panel#2入板訊號
      MPS
      AND     T221
      RST     M5121  ; 回上位Panel#2入板訊號
      MPP
      OUT     T221 K30
4082  LD      M5122  ; 回上位Panel#3入板訊號
      MPS
      AND     T222
      RST     M5122  ; 回上位Panel#3入板訊號
      MPP
      OUT     T222 K30
4091  LD      M5123  ; 回上位Panel#4入板訊號
      MPS
      AND     T223
      RST     M5123  ; 回上位Panel#4入板訊號
      MPP
      OUT     T223 K30
4100  LD      M5125  ; 回上位Panel#1出板訊號
      MPS
      AND     T225
      RST     M5125  ; 回上位Panel#1出板訊號
      MPP
      OUT     T225 K30
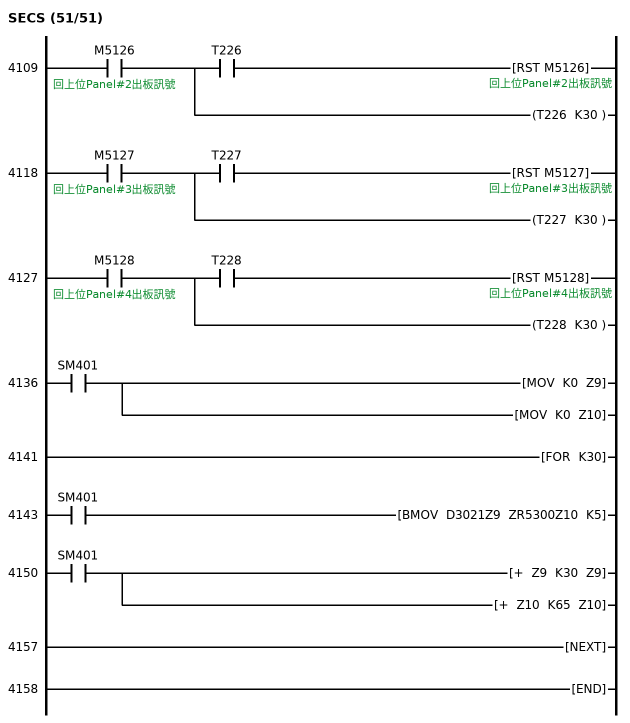
4109  LD      M5126  ; 回上位Panel#2出板訊號
      MPS
      AND     T226
      RST     M5126  ; 回上位Panel#2出板訊號
      MPP
      OUT     T226 K30
4118  LD      M5127  ; 回上位Panel#3出板訊號
      MPS
      AND     T227
      RST     M5127  ; 回上位Panel#3出板訊號
      MPP
      OUT     T227 K30
4127  LD      M5128  ; 回上位Panel#4出板訊號
      MPS
      AND     T228
      RST     M5128  ; 回上位Panel#4出板訊號
      MPP
      OUT     T228 K30
4136  LD      SM401
      MOV     K0 Z9
      MOV     K0 Z10
4141  FOR     K30
4143  LD      SM401
      BMOV    D3021Z9 ZR5300Z10 K5
4150  LD      SM401
      +       Z9 K30 Z9
      +       Z10 K65 Z10
4157  NEXT
4158  END
END_PROGRAM

// device comments not shown above
X6E  ; 冷卻段排風風車過載
X90  ; 冷卻段強制排氣風車變頻器運轉
X9C  ; 第二槽IR4低溫異常
X9D  ; 第二槽IR4超溫異常
X9E  ; 第二槽IR4超溫防止器異常
X0B9  ; 第三槽IR6低溫異常
X0BA  ; 第三槽IR6超溫異常
X0BB  ; 第三槽IR6超溫防止器異常
Y102  ; 上游<--印刷(3)允許入料
Y103  ; 上游<--印刷(4)允許入料
Y106  ; 下游SP
Y107  ; 下游SP
Y125  ; 第二槽IR4電磁開關
Y126  ; 第三槽IR6電磁開關
Y12D  ; 出料黏塵輪升降電磁閥
Y12E  ; 入出口(接駁輪)吹氣電磁閥(關)
M9  ; 回路3
M10  ; 入出口(接駁輪)吹氣電磁閥 M
M17  ; 出料黏塵輪自動升降 RY
M18  ; 出料黏塵輪上升RY
M19  ; 出料黏塵輪下降RY
M34  ; 第5槽電熱溫度到
M35  ; 第6槽電熱溫度到
M36  ; 第7槽電熱溫度到
M37  ; 第8槽電熱溫度到
M38  ; 第9槽電熱溫度到
M39  ; 第10槽電熱溫度到
M43  ; 第14槽電熱溫度到
M50  ; 第2槽IR4溫度到
M51  ; 第3槽IR6溫度到
M53  ; 第9槽IR9溫度到
M54  ; 第10槽IR10溫度到
M55  ; 第11槽IR11溫度到
M56  ; 第12槽IR12溫度到
M57  ; 第13槽IR13溫度到
M58  ; 第14槽IR14溫度到
M70  ; 印刷有板偵測光電1
M71  ; 印刷有板偵測光電2
M72  ; 印刷有板偵測光電3
M73  ; 印刷有板偵測光電4
M90  ; 輸送暫停
M113  ; 第5槽風車5-GP
M114  ; 第5槽電熱5-GP
M115  ; 第5槽IR5-GP
M116  ; 第6槽風車6-GP
M117  ; 第6槽電熱6-GP
M118  ; 第6槽IR6-GP
M119  ; 第7槽風車7-GP
M120  ; 第7槽電熱7-GP
M121  ; 第7槽IR7-GP
M122  ; 第8槽風車8-GP
M123  ; 第8槽電熱8-GP
M124  ; 第8槽IR8-GP
M125  ; 第9槽風車9-GP
M126  ; 第9槽電熱9-GP
M127  ; 第9槽IR9-GP
M128  ; 第10槽風車10-GP
M129  ; 第10槽電熱10-GP
M130  ; 第10槽IR10-GP
M131  ; 第11槽風車11-GP
M132  ; 第11槽電熱11-GP
M133  ; 第11槽IR11-GP
M134  ; 第12槽風車12-GP
M135  ; 第12槽電熱12-GP
M136  ; 第12槽IR12-GP
M137  ; 第13槽風車13-GP
M138  ; 第13槽電熱13-GP
M139  ; 第13槽IR13-GP
M140  ; 第14槽風車14-GP
M141  ; 第14槽電熱14-GP
M142  ; 第14槽IR14-GP
M146  ; 熱排風風車 GP
M147  ; 熱排風風車高速 GP
M152  ; 出料黏塵輪上升 GP
M161  ; 第2槽IR4-GP
M162  ; 第3槽IR6-GP
M165  ; IR4-PLS
M166  ; IR6-PLS
M175  ; 第五槽風車電磁開關 M
M176  ; 第六槽風車電磁開關 M
M177  ; 第七槽風車電磁開關 M
M178  ; 第八槽風車電磁開關 M
M179  ; 第九槽風車電磁開關 M
M180  ; 第十槽風車電磁開關 M
M181  ; 第十一槽風車電磁開關 M
M182  ; 第十二槽風車電磁開關 M
M183  ; 第十三槽風車電磁開關 M
M184  ; 第十四槽風車電磁開關 M
M191  ; IR4-RY
M192  ; IR6-RY
M213  ; 風車5-PLS
M214  ; 電熱5-PLS
M215  ; IR5-PLS
M216  ; 風車6-PLS
M217  ; 電熱6-PLS
M218  ; IR6-PLS
M219  ; 風車7-PLS
M220  ; 電熱7-PLS
M221  ; IR7-PLS
M222  ; 風車8-PLS
M223  ; 電熱8-PLS
M224  ; IR8-PLS
M225  ; 風車9-PLS
M226  ; 電熱9-PLS
M227  ; IR9-PLS
M246  ; 熱排風風車 PLS
M247  ; 熱排風風車二段速 PLS
M252  ; 出料黏塵輪上升 PLS
M275  ; 第五槽電熱電磁開關 M
M276  ; 第六槽電熱電磁開關 M
M277  ; 第七槽電熱電磁開關 M
M278  ; 第八槽電熱電磁開關 M
M279  ; 第九槽電熱電磁開關 M
M280  ; 第十槽電熱電磁開關 M
M281  ; 第十一槽電熱電磁開關 M
M282  ; 第十二槽電熱電磁開關 M
M283  ; 第十三槽電熱電磁開關 M
M284  ; 第十四槽電熱電磁開關 M
M299  ; 維修保養畫面PB
M313  ; 風車5-RY
M314  ; 電熱5-RY
M315  ; IR5-RY
M316  ; 風車6-RY
M317  ; 電熱6-RY
M318  ; IR6-RY
M319  ; 風車7-RY
M320  ; 電熱7-RY
M321  ; IR7-RY
M322  ; 風車8-RY
M323  ; 電熱8-RY
M324  ; IR8-RY
M325  ; 風車9-RY
M326  ; 電熱9-RY
M327  ; IR9-RY
M328  ; 風車10-RY
M329  ; 電熱10-RY
M330  ; IR10-RY
M331  ; 風車11-RY
M332  ; 電熱11-RY
M333  ; IR11-RY
M334  ; 風車12-RY
M335  ; 電熱12-RY
M336  ; IR12-RY
M337  ; 風車13-RY
M338  ; 電熱13-RY
M339  ; IR13-RY
M340  ; 風車14-RY
M341  ; 電熱14-RY
M342  ; IR14-RY
M346  ; 熱排風風車 RY
M347  ; 熱排風風車二段速RY
M352  ; 出料黏塵輪上升 RY
M363  ; 出料黏塵輪升降電磁閥 M
M366  ; 熱排風風車運轉 M
M367  ; 熱排風風車二段速 M
M379  ; 第九槽IR9電磁開關 M
M380  ; 第十槽IR10電磁開關 M
M381  ; 第十一槽IR11電磁開關 M
M382  ; 第十二槽IR12電磁開關 M
M383  ; 第十三槽IR13電磁開關 M
M384  ; 第十四槽IR14電磁開關 M
M408  ; 啟動 8
M412  ; 啟動 12
M419  ; 啟動 19
M420  ; 啟動 20
M421  ; 啟動 21
M422  ; 啟動 22
M423  ; 啟動 23
M424  ; 啟動 24
M425  ; 啟動 25
M426  ; 啟動 26
M427  ; 啟動 27
M428  ; 啟動 28
M429  ; 啟動 29
M430  ; 啟動 30
M432  ; 啟動 32
M433  ; 啟動 33
M434  ; 啟動 34
M435  ; 啟動 35
M436  ; 啟動 36
M437  ; 啟動 37
M438  ; 啟動 38
M439  ; 啟動 39
M440  ; 啟動 40
M441  ; 啟動 41
M442  ; 啟動 42
M443  ; 啟動 43
M444  ; 啟動 44
M445  ; 啟動 45
M446  ; 啟動 46
M447  ; 啟動 47
M448  ; 啟動 48
M449  ; 啟動 49
M450  ; 啟動 50
M451  ; 啟動 51
M452  ; 啟動 52
M453  ; 啟動 53
M454  ; 啟動 54
M455  ; 啟動 55
M456  ; 啟動 56
M457  ; 啟動 57
M458  ; 啟動 58
M459  ; 啟動 59
M460  ; 啟動 60
M461  ; 啟動 61
M462  ; 啟動 62
M463  ; 啟動 63
M489  ; 下游連線連鎖 RY
M497  ; TEST1(HI)
M506  ; 停止 6
M509  ; 停止 9
M513  ; 停止 13
M514  ; 停止 14
M515  ; 停止 15
M516  ; 停止 16
M517  ; 停止 17
M518  ; 停止 18
M524  ; 停止 24
M525  ; 停止 25
M526  ; 停止 26
M527  ; 停止 27
M528  ; 停止 28
M532  ; 停止 32
M533  ; 停止 33
M534  ; 停止 34
M535  ; 停止 35
M536  ; 停止 36
M537  ; 停止 37
M538  ; 停止 38
M539  ; 停止 39
M540  ; 停止 40
M541  ; 停止 41
M542  ; 停止 42
M543  ; 停止 43
M544  ; 停止 44
M545  ; 停止 45
M546  ; 停止 46
M547  ; 停止 47
M548  ; 停止 48
M549  ; 停止 49
M550  ; 停止 50
M551  ; 停止 51
M552  ; 停止 52
M553  ; 停止 53
M554  ; 停止 54
M555  ; 停止 55
M556  ; 停止 56
M557  ; 停止 57
M558  ; 停止 58
M559  ; 停止 59
M560  ; 停止 60
M561  ; 停止 61
M562  ; 停止 62
M563  ; 停止 63
M800  ; 緊急停止迴圈資料
M4170  ; [PPID]  配方搜尋比對OK_配方可
M4541  ; 入料片數到達
M6013  ; 設備生產訊號收集-配方程式安裝開
M6014  ; 設備生產訊號收集-配方程式安裝結
M6059  ; Host刪除配方
M6060  ; Host刪除配方完成
M6134  ; 三色燈狀態改變
M6140  ; 要求上位回讀工單板號右爐
M6141  ; 要求上位回讀工單右爐
M6142  ; 三色黃燈
M6231  ; 上位要儲存配方
M6300  ; 緊急停止開關異常
M6301  ; 逆相繼電器異常
M6302  ; 入口卡板異常
M6303  ; 出口卡板異常
M6304  ; UV門防止打開開關異常
M6305  ; 上排風風車過載
M6306  ; 下排風風車過載
M6307  ; 安定器冷卻風扇過載
M6308  ; 第一燈溫度異常
M6309  ; 下燈1點燈異常
M6310  ; 下燈2點燈異常
M6311  ; 上燈1點燈異常
M6312  ; 上燈2點燈異常
M6313  ; 變頻機異常
M6314  ; 出料連線異常
M6315  ; 爐內限制數量異常
M6316  ; PLC Low Battery
M6317  ; 進氣冷卻風扇過載
M6318  ; 燈箱冷卻風扇過載
M6319  ; 輸送運轉未點燈警報
M6320  ; 點燈中輸送停止未運轉
M6321  ; 板子有進沒出m231沒滅
M6322  ; 輸送馬達過載異常
M6323  ; 網偏前警報
M6324  ; 網偏後警報
M6325  ; 燈箱冷卻風扇過載
M6326  ; 進氣冷卻風扇過載
M6327  ; 網偏警報熄燈計時
M6328  ; 第二燈溫度異常
M6330  ; UV點燈後30秒不可選擇提示
M6331  ; 下燈1管保養時間到達
M6332  ; 下燈2管保養時間到達
M6333  ; 上燈1管保養時間到達
M6334  ; 上燈2管保養時間到達
M6335  ; 滾輪保養時間到達
M6336  ; 輸送馬達過載異常
M6339  ; 節能省電啟動
M6340  ; 出口卡板異常
M6344  ; 安全門開啟時熄燈選擇    (on熄燈)
M6345  ; 卡板熄燈
M6349  ; 下燈1   點燈失敗
M6350  ; 下燈2   點燈失敗
M6351  ; 上燈1   點燈失敗
M6352  ; 上燈2   點燈失敗
T74  ; 第五槽電熱低溫延遲60S
T75  ; 第六槽電熱低溫延遲60S
T76  ; 第七槽電熱低溫延遲60S
T77  ; 第八槽電熱低溫延遲60S
T78  ; 第九槽電熱低溫延遲60S
T79  ; 第十槽電熱低溫延遲60S
T80  ; 第十一槽電熱低溫延遲60S
T81  ; 第十二槽電熱低溫延遲60S
T82  ; 第十三槽電熱低溫延遲60S
T83  ; 第十四槽電熱低溫延遲60S
T90  ; 第二槽IR4低溫延遲60S
T91  ; 第三槽IR6低溫延遲60S
T93  ; 第九槽IR9低溫延遲60S
T94  ; 第十槽IR10低溫延遲60S
T95  ; 第十一槽IR11低溫延遲60S
T96  ; 第十二槽IR12低溫延遲60S
T97  ; 第十三槽IR13低溫延遲60S
T98  ; 第十四槽IR14低溫延遲60S
D110  ; DA輸出值
D112  ; DA1輸出放大值
D160  ; SECS_上位傳數量(BIN)
D230  ; SPM3-Address
D231  ; SPM3-BaudRate
D232  ; SPM3-StopBit
D233  ; SPM3-Mode
D234  ; SPM3-PT_Primary
D236  ; SPM3-PT_Secondary
D237  ; SPM3-CT_Primary
D238  ; SPM3-CT_Secondary
D258  ; 黏塵輪上升時間
D259  ; 黏塵輪下降時間
D264  ; 出料黏塵輪上升時間*10
D266  ; 出料黏塵輪下降時間*10
D364  ; DA2
D404  ; outside DA-CH3  收捲    0~10V
D406  ; outside DA-CH4
D410  ; 放捲傳動正常值
D412  ; 輸送速度/10(SV)
D420  ; 放捲HI設定
D422  ; 放捲HI值
D424  ; 放捲高速
D426  ; 高速(32bit)
D428  ; 放捲傳動高速值
D440  ; 放捲LO設定
D442  ; 放捲LO值
D444  ; 放捲低速
D446  ; 低速(32bit)
D448  ; 放捲傳動低速值
D500  ; 輸送速度(SV)
D501  ; 輸送速度(SV)
D801  ; TO溫控器設定值IR1
D802  ; TO溫控器設定值IR2
D803  ; TO溫控器設定值TC02
D804  ; TO溫控器設定值IR3
D805  ; TO溫控器設定值TC03
D806  ; TO溫控器設定值IR4
D807  ; TO溫控器設定值TC04
D808  ; TO溫控器設定值IR5
D809  ; TO溫控器設定值IR6
D5090  ; 前次四色燈藍燈狀態
D5091  ; 目前四色燈藍燈狀態
D5300  ; 當前使用配方Recipe NO.
D5350  ; K
D5351  ; L
D5352  ; M
D5353  ; N
D5354  ; O
D5355  ; P
D5356  ; Q
D5357  ; R
D5358  ; S
D5359  ; T
D5380  ; IR1-SV
D5381  ; IR2-SV
D5382  ; 電熱2-SV
D5383  ; IR3-SV
D5384  ; IR4-SV
D5385  ; 電熱3-SV
D5386  ; IR5-SV
D5387  ; IR6-SV
D5388  ; 電熱4-SV
D5389  ; IR7-SV
D5390  ; IR8-SV
D5399  ; 輸送速度-SV
D5409  ; 配方組別
D10070  ; 比對START字串
D10071  ; 比對STOP字串
D10072  ; 比對PP_SELECT字串
D10074  ; 比對配方名稱為零可儲存位址
D10076  ; 名稱有一樣的是更新=50要新增
D10077  ; 比對PAUSE字串
D10078  ; 比對RESUME字串
D10081  ; 上位下配方比對結果
D10083  ; 上位下的組別右門(比對出來的)
D10084  ; 名稱GO-LOCAL比對結果
D10085  ; 名稱PPID比對結果
D10086  ; 上位下配方比對結果
D10087  ; 上位下的組別左門(比對出來的)
D10661  ; SECS_上位下PAUSE指令
D10662  ; SECS_上位下PAUSE指令
D13610  ; 查詢配方內容:IR7-SV
D13611  ; 查詢配方內容:IR8-SV
D13620  ; 電熱#1溫度設定SV(FLT)
D13621  ; 電熱#1溫度設定SV(FLT)
D13622  ; IR#1溫度設定SV(FLT)
D13623  ; IR#1溫度設定SV(FLT)
D13624  ; IR#2溫度設定SV(FLT)
D13625  ; IR#2溫度設定SV(FLT)
D13626  ; 電熱#2溫度設定SV(FLT)
D13627  ; 電熱#2溫度設定SV(FLT)
D13628  ; IR#3溫度設定SV(FLT)
D13629  ; IR#3溫度設定SV(FLT)
D13630  ; IR#4溫度設定SV(FLT)
D13631  ; IR#4溫度設定SV(FLT)
D13632  ; 電熱#3溫度設定SV(FLT)
D13633  ; 電熱#3溫度設定SV(FLT)
D13634  ; IR#5溫度設定SV(FLT)
D13635  ; IR#5溫度設定SV(FLT)
D13636  ; IR#6溫度設定SV(FLT)
D13637  ; IR#6溫度設定SV(FLT)
D13638  ; 電熱#4溫度設定SV(FLT)
D13639  ; 電熱#4溫度設定SV(FLT)
D13640  ; IR#7溫度設定SV(FLT)
D13641  ; IR#7溫度設定SV(FLT)
D13642  ; IR#8溫度設定SV(FLT)
D13643  ; IR#8溫度設定SV(FLT)
D13645  ; 輸送速度設定SV(FLT)
ZR2173  ; 查詢配方內容:IR8-FLT
ZR5201  ; SECS_上位配方NO.01
ZR5300  ; PPID(Name)
ZR5302  ; PPID(Name)
ZR5341  ; 變更狀態
ZR10001  ; IR1-SV
ZR10002  ; IR2-SV
ZR10003  ; 電熱2-SV
ZR10004  ; IR3-SV
ZR10005  ; IR4-SV
ZR10006  ; 電熱3-SV
ZR10007  ; IR5-SV
ZR10008  ; IR6-SV
ZR10009  ; 電熱4-SV
ZR10010  ; IR7-SV
ZR10011  ; IR8-SV
ZR10020  ; 輸送速度-SV
